{attribute addProperty BoxType "EL2912-0000-0016"}
{attribute addProperty Id "FSOEAT %Q*FSOE_3A505F92486"}
{attribute addProperty CRC "1772735418"}
{attribute addProperty SizeInBites "48"}
{attribute addProperty SizeInBytes "6"}
TYPE FSoE_Outputs_69A9CBBA :
STRUCT
	{attribute addProperty Name "FSOE"}
	FSOE AT %Q* : FSOE_3A505F92;
END_STRUCT
END_TYPE

(* stored: Version 1.2.0.0, ProductVersion 3.1.4024.9
   DUT FSoE_Outputs_69A9CBBA: Id {3a8d3dcf-04ec-4630-a66f-88dfd7fd894f} *)
